Staubli VAL3: refreshDynamic.pgx

program refreshDynamic()
begin
    // DO NOT CHANGE
  nRefresh=clock()
  use:bUseRefresh=false
  //
  // ADD HERE
  //
end
